(* IEC 61131-3 sources: moqui-plc/simatic-ax/src/moqui/framework/src/main/org/moqui/device, 20 files *)

(* ---- ActuatorActuationType.st ---- *)
TYPE ActuatorActuationType : (
    SingleActuation, (* Single Actuation: Uses enable output only *)
    DoubleActuation, (* Double Actuation: enable/disable are pulses *)
    DoubleActuationNoRetain (* Double Actuation: enable/disable are levels *)
); END_TYPE

(* ---- ActuatorFeedbackType.st ---- *)
TYPE ActuatorFeedbackType : (
	WithoutFeedback, (* No feedback *)
    SingleDisableFeedback, (* Single Deactivation Feedback: Only disabledSensor *)
    SingleEnableFeedback, (* Single Activation Feedback: Only enabledSensor *)
	DoubleFeedback (* Double Feedback: Both sensors *)
); END_TYPE

(* ---- ActuatorModel.st ---- *)
TYPE ActuatorModel : (
	ABBACH580, (* ABB ACH580 *)
	CTM700, (* Control Techniques CM700 *)
	DanfossFC102, (* Danfoss FC102 *)
	ABBPSTX (* ABB PSTX SoftStarter *)
	(* etc. *)
); END_TYPE

(* ---- ActuatorStatus.st ---- *)
TYPE ActuatorStatus : (
	Disabled, (* Stable *)
	EnablePhase, (* Unstable *)
	Enabled, (* Stable *)
	DisablePhase (* Unstable *)
); END_TYPE

(* ---- ActuatorType.st ---- *)
TYPE ActuatorType : (
  OnOff, (* Fallback value *)
  Contactor,
  SoftStarter,
  Vfd, (* Frequency converter / Inverter drive *)
  PneumaticCylinder,
  PneumaticValve,
  HydraulicCylinder,
  HydraulicValve,
  Damper,
  SolenoidValve
  (* etc. *)
); END_TYPE

(* ---- DeviceConfigCmdType.st ---- *)
(* After each creation, saving or deletion of device config it will be necessary to reload the config list with the Init command. *)
TYPE DeviceConfigCmdType : (
    Init, (* Init the recipe management component *)
	Create,
    Save,
	Load,
	Delete,
	Reset
); END_TYPE

(* ---- DeviceConfigMgmtStatus.st ---- *)
TYPE DeviceConfigMgmtStatus : (
    Idle,
	Init,
	Resetting,
    Check,
    Load,
    WaitLoad,
    WaitProcessing,
    IncrementIndex,
    Completed,
    Error
); END_TYPE

(* ---- DriveControlWord.st ---- *)
(* Drive control words *)
(* Relevant control word for start, stop and reset commands *)
TYPE DriveControlWord : (
	(* ABB ACS580, ACH580 drive *)
	ABBACH580Reset,
	ABBACH580Stop,
	ABBACH580Start,
	(* Control Techniques M600 drive *)
	CTM600Reset,
	CTM600Stop,
	CTM600Start,
	(* Danfoss FC102 drive *)
	DanfossFC102Reset,
	DanfossFC102Stop,
	DanfossFC102Start
); END_TYPE

(* ---- EdgeTriggerStatus.st ---- *)
TYPE EdgeTriggerStatus : (
	Dormant,
	Executing,
	Done,
	Aborting,
	Aborted,
	Resetting,
	Error
); END_TYPE

(* ---- LevelCtrlStatus.st ---- *)
TYPE LevelCtrlStatus : (
	Dormant,
	Executing,
	Done,
	Aborting,
	Resetting,
	Error
); END_TYPE

(* ---- OperatingMode.st ---- *)
TYPE OperatingMode : (
	Init,
	Run
); END_TYPE

(* ---- RampType.st ---- *)
TYPE RampType : (
    Linear, // Linear ramp.
    SShaped, // S-Shaped ramp.
    Exponential, // Exponential ramp
    Custom // Custom-defined ramp function
); END_TYPE

(* ---- SpeedSetpointLevel.st ---- *)
(* Constants are defined to represent the different speed levels required by a motor.
 * Alternatively, the speed setpoint/reference can be defined as a continuous analog output.
 * It is possible to apply the same logic to other variables such as:
 *     acceleration/deceleration, torque, etc.
 *)
TYPE SpeedSetpointLevel : (
	ZeroSpeed,
	NominalSpeed,
	MinSpeed,
	MaxSpeed,
	JoggingSpeed,
	SafelyLimitedSpeed
	(* etc. *)
); END_TYPE

(* ---- ParseRecipeTime.st ---- *)
USING System.Strings;

FUNCTION ParseRecipeTime : TIME
	VAR_INPUT
		value : STRING;
	END_VAR
	VAR_TEMP
		normalizedValue : STRING[32];
		numberText : STRING[16];
		unitText : STRING[2];
		valueLength : INT;
		magnitude : DINT;
		position : DINT;
	END_VAR

	normalizedValue := value;
	valueLength := LengthOf(normalizedValue);

	IF (valueLength >= INT#5) AND (Substring(normalizedValue, INT#1, INT#5) = 'TIME#') THEN
		normalizedValue := Substring(normalizedValue, INT#6, valueLength - INT#5);
	ELSIF (valueLength >= INT#2) AND (Substring(normalizedValue, INT#1, INT#2) = 'T#') THEN
		normalizedValue := Substring(normalizedValue, INT#3, valueLength - INT#2);
	END_IF;

	valueLength := LengthOf(normalizedValue);
	IF valueLength <= INT#0 THEN
		RETURN;
	END_IF;

	IF (valueLength >= INT#2) AND (Substring(normalizedValue, valueLength - INT#1, INT#2) = 'ms') THEN
		unitText := 'ms';
		numberText := Substring(normalizedValue, INT#1, valueLength - INT#2);
	ELSIF (valueLength >= INT#1) THEN
		unitText := Substring(normalizedValue, valueLength, INT#1);
		numberText := Substring(normalizedValue, INT#1, valueLength - INT#1);
	END_IF;

	magnitude := ParseRecipeDInt(numberText);
	IF magnitude <= DINT#0 THEN
		RETURN;
	END_IF;

	CASE unitText OF
		'ms' :
			FOR position := DINT#1 TO magnitude DO
				ParseRecipeTime := ParseRecipeTime + T#1ms;
			END_FOR;
		's' :
			FOR position := DINT#1 TO magnitude DO
				ParseRecipeTime := ParseRecipeTime + T#1s;
			END_FOR;
		'm' :
			FOR position := DINT#1 TO magnitude DO
				ParseRecipeTime := ParseRecipeTime + T#1m;
			END_FOR;
		'h' :
			FOR position := DINT#1 TO magnitude DO
				ParseRecipeTime := ParseRecipeTime + T#1h;
			END_FOR;
	END_CASE;
END_FUNCTION

(* ---- Actuator.st ---- *)
(*
 * Generic binary actuator control system/automata, including mechanisms diagnostics.
 * In nominal conditions, a binary actuator has only two stable equilibrium states: Disabled, Enabled.
 * It also has two unstable transient states: EnablePhase, DisablePhase.
 * The remainder are inadmissible states that must be detected based on timing conditions.
 * Nominal trajectory in the state space, i.e. the evolution of the state in nominal working conditions:
 *     Disabled --> EnablePhase --> Enabled --> DisabledPhase --> back to Disabled
 * Admissible states transitions:
 *     EnablePhase --> DisablePhase, DisablePhase --> EnablePhase
 *
 * Handshake-based actuator control via VAR_IN_OUT.
 * This function block utilizes a Request/Acknowledge (Handshake) mechanism
 * through VAR_IN_OUT variables to manage asynchronous device operations.
 *
 * Usage Logic:
 *  - The caller sets the 'enableRequest' variable to TRUE to initiate the process.
 *  - The FB monitors this variable and attempts to enable the physical device.
 *  - Upon successful activation, the FB internally resets 'enableRequest' to FALSE.
 *
 * Sequencing and diagnostics:
 *  - Sequencing: By monitoring the falling edge of the request variable (Request -> FALSE),
 *    the application logic can deterministically trigger the next step in a sequence
 *    without relying on timers or intermediate state flags.
 *  - Real-Time diagnostics: If the request remains TRUE beyond a defined timeout period,
 *    it indicates a failure in the handshake (e.g., hardware interlock or communication error).
 *    This allows for immediate error detection (machineError) and prevents the
 *    sequence from advancing in an unsafe state.
 *
 * Note:
 * Since the variable is passed by reference (VAR_IN_OUT), both the caller and
 * the FB share the same memory location, ensuring atomic-like synchronization of the command status.
 * This mechanism is used to allow sequencing of the start/stop phases in the presence of a group of devices.
 *
 *)
FUNCTION_BLOCK Actuator
	(* Request/Ack commands *)
	VAR_IN_OUT
	    enableRequest : BOOL;
	    disableRequest : BOOL;
	END_VAR
	VAR_INPUT
		(* Actuator metadata for logging purpose *)
		actuatorId : STRING;
		actuatorName : STRING;
	  	actuationType : ActuatorActuationType;
		feedbackType : ActuatorFeedbackType;
		model : ActuatorModel;
	    operationType : OperatingMode := OperatingMode#Run;
		(* Clock for diagnosis and fault detection under static and dynamic conditions *)
	    clock : BOOL;
		(* Time limit for the enable/disable phase *)
	    enableTime : UINT;
	    disableTime : UINT;
		(* Preset/Reset *)
	    enablePreset : BOOL := FALSE;
	    (* Enable diagnostics *)
	    diagnosticsEnable : BOOL := TRUE;
	END_VAR
	VAR_INPUT
		(* Actuator status sensors *)
	    enabledSensor : BOOL;
	    disabledSensor : BOOL;
		(* External fault signal (e.g. motor branch-circuit protection, thermal relay) *)
		externalFault : BOOL;
		(* Optional parameters  *)
	  	referenceValue : REAL;
	  	feedback : REAL;
	END_VAR
	VAR_OUTPUT
		(* Diagnostics and fault signals *)
	    fault : BOOL;
	    actuatorFault : BOOL;
	    enabledSensorFault : BOOL;
	    disabledSensorFault : BOOL;
	    notInitialized : BOOL;
		(* Logger name for centralized signal management *)
		loggerName : STRING;
	END_VAR
	VAR_OUTPUT
		(* Output signals *)
		enable : BOOL;
	    disable : BOOL;
	END_VAR
	VAR
	    status : ActuatorStatus;
	    timer : UINT;
	    timeout : BOOL;
		(* Internal logical feedback signals (derived from external sensors and/or state + timeout). *)
		enabled : BOOL;
		disabled : BOOL;
		(* Logger facade *)
		logger : LoggerFacade;
	END_VAR

	(* Initialization handler *)
	IF operationType = OperatingMode#Init THEN
		(* Args validation *)
		IF (actuatorId = '' AND actuatorName = '') THEN
			notInitialized := TRUE;
			RETURN;
		END_IF;

		(* Logger facade init *)
		loggerName := actuatorName;
		IF loggerName = '' THEN
			loggerName := actuatorId;
		END_IF;
		logger.enable := TRUE; logger.loggerName := loggerName;

		logger(message := 'Actuator initialization.', level := LogLevel#DEBUG);

		(* Pre-elaborations for initialization (polymorphism on feedback typology). *)
		CASE feedbackType OF
			ActuatorFeedbackType#DoubleFeedback :
				enabled := enabledSensor;
				disabled := disabledSensor;

			ActuatorFeedbackType#SingleEnableFeedback :
				enabled := enabledSensor;
				disabled := NOT enabled;

			ActuatorFeedbackType#SingleDisableFeedback :
				disabled := disabledSensor;
				enabled := NOT disabled;

			ActuatorFeedbackType#WithoutFeedback :
				enabled := enablePreset;
				disabled := NOT enabled;
		END_CASE;

		enableRequest := FALSE;
		disableRequest := FALSE;

	    IF enablePreset THEN
			logger(message := 'Actuator preset to enabled status.', level := LogLevel#DEBUG);
			enable := TRUE;
			timer := enableTime;

			IF enabled THEN
				status := ActuatorStatus#Enabled;
				notInitialized := FALSE;
			ELSE
				status := ActuatorStatus#EnablePhase;
	            notInitialized := TRUE;
			END_IF;
	    ELSE
			logger(message := 'Actuator preset to disabled status.', level := LogLevel#DEBUG);
			enable := FALSE;
			timer := disableTime;

			IF disabled THEN
	            status := ActuatorStatus#Disabled;
	            notInitialized := FALSE;
	        ELSE
	            status := ActuatorStatus#DisablePhase;
	            notInitialized := TRUE;
	        END_IF;
		END_IF;
	END_IF;

	IF notInitialized THEN logger(message := 'Actuator not initialized.', level := LogLevel#ERROR); END_IF;

	logger(message := 'Running actuator.', level := LogLevel#DEBUG);

	(* Clock handler for diagnosis oriented timing *)
	IF clock AND (timer > UINT#0) THEN
	    timer := timer - UINT#1;
	END_IF;

	(* Timeout computation *)
	timeout := (timer = UINT#0);

	(* Pre-elaborations for feedback polymorphism. *)
	CASE feedbackType OF
		ActuatorFeedbackType#DoubleFeedback :
			enabled := enabledSensor;
			disabled := disabledSensor;

		ActuatorFeedbackType#SingleDisableFeedback :
			disabled := disabledSensor;
			enabled := (NOT disabled) AND ((status = ActuatorStatus#Enabled)
				OR ((status = ActuatorStatus#EnablePhase) AND timeout));

		ActuatorFeedbackType#SingleEnableFeedback :
			enabled := enabledSensor;
			disabled := (NOT enabled) AND ((status = ActuatorStatus#Disabled)
				OR ((status = ActuatorStatus#DisablePhase) AND timeout));

		ActuatorFeedbackType#WithoutFeedback :
			enabled := (status = ActuatorStatus#Enabled) OR ((status = ActuatorStatus#EnablePhase) AND timeout);
			disabled := (status = ActuatorStatus#Disabled) OR ((status = ActuatorStatus#DisablePhase) AND timeout);
	END_CASE;

	(* Generic actuator FSM implementation. *)
	CASE status OF
		ActuatorStatus#Disabled :
			logger(message := 'Actuator disabled.', level := LogLevel#DEBUG);
			disableRequest := FALSE;

			IF enableRequest THEN
				logger(message := 'The actuator received an enable request.', level := LogLevel#DEBUG);
				enable := TRUE;
				timer := enableTime;
				status := ActuatorStatus#EnablePhase;
			END_IF;

		ActuatorStatus#EnablePhase :
			logger(message := 'Actuator in the enabling phase.', level := LogLevel#DEBUG);

			(* Admissible transition: EnablePhase --> DisablePhase *)
			IF disableRequest THEN
				logger(message := 'The actuator received a disable request.', level := LogLevel#DEBUG);
				enableRequest := FALSE;
				enable := FALSE;
				timer := disableTime;
				status := ActuatorStatus#DisablePhase;
			ELSIF enabled THEN
				(* End of the enable phase, by feedback or by timeout in no-feedback typology. *)
				enableRequest := FALSE;
				timer := UINT#0;
				status := ActuatorStatus#Enabled;
			END_IF;

		ActuatorStatus#Enabled :
			logger(message := 'Actuator enabled.', level := LogLevel#DEBUG);
			enableRequest := FALSE;

			IF disableRequest THEN
				logger(message := 'The actuator received a disable request.', level := LogLevel#DEBUG);
				enable := FALSE;
				timer := disableTime;
				status := ActuatorStatus#DisablePhase;
			END_IF;

		ActuatorStatus#DisablePhase :
			logger(message := 'Actuator in the disabling phase.', level := LogLevel#DEBUG);

			(* Admissible transition: DisablePhase --> EnablePhase *)
			IF enableRequest THEN
					logger(message := 'The actuator received an enable request.', level := LogLevel#DEBUG);
					disableRequest := FALSE;
					enable := TRUE;
					timer := enableTime;
					status := ActuatorStatus#EnablePhase;
			ELSIF disabled THEN
				(* End of the disable phase, by feedback or by timeout in no-feedback typology. *)
				disableRequest := FALSE;
				timer := UINT#0;
				status := ActuatorStatus#Disabled;
			END_IF;
	END_CASE;

	(*
	 * Diagnostics handler.
	 * Generation of diagnosis information and fault signals: Detectable faults in dynamic and static conditions.
	 *)
	disabledSensorFault := diagnosticsEnable AND (
	    (NOT enable AND NOT disabled AND NOT enabled
		OR enable AND disabled AND enabled) AND timeout);
	enabledSensorFault := diagnosticsEnable AND (
	    (NOT enable AND disabled AND enabled
		OR enable AND NOT disabled AND NOT enabled) AND timeout);
	actuatorFault := diagnosticsEnable AND (
	    (NOT enable AND NOT disabled AND enabled
		OR enable AND disabled AND NOT enabled) AND timeout);
	fault := disabledSensorFault OR enabledSensorFault OR actuatorFault OR externalFault;
	(* Log faults *)
	IF fault THEN logger(message := 'Fault diagnostics:', level := LogLevel#ERROR); END_IF;
	IF disabledSensorFault THEN logger(message := 'Disabled sensor fault.', level := LogLevel#ERROR); END_IF;
	IF enabledSensorFault THEN logger(message := 'Enabled sensor fault.', level := LogLevel#ERROR); END_IF;
	IF actuatorFault THEN logger(message := 'Actuator fault.', level := LogLevel#ERROR); END_IF;
	IF externalFault THEN logger(message := 'External fault (e.g: Motor branch-circuit protection).', level := LogLevel#ERROR); END_IF;

	(* Post-elaborations for actuation polymorphism. *)
	CASE actuationType OF
		ActuatorActuationType#SingleActuation :
			(* Nothing to do, just use enable *);
		ActuatorActuationType#DoubleActuation :
			disable := NOT enable;
		ActuatorActuationType#DoubleActuationNoRetain :
			enable := enable AND (status = ActuatorStatus#EnablePhase);
			disable := NOT enable AND (status = ActuatorStatus#DisablePhase);
	END_CASE;
	END_FUNCTION_BLOCK

(* ---- DeviceConfigCmds.st ---- *)
USING Siemens.Simatic.S71500.FileAccess;
USING System.Strings;

FUNCTION_BLOCK DeviceConfigCmds
	VAR_EXTERNAL CONSTANT
		DEVICE_CONFIG_LIST_MAX_SIZE : UINT;
		defaultConfigType : STRING;
		deviceConfigStoragePath : STRING;
	END_VAR
	VAR_EXTERNAL
		dev : DeviceFacade;
	END_VAR
	VAR_INPUT
	    configType : STRING := defaultConfigType; (* If empty, set default device config type *)
		(*
	     * The default file name of a recipe is: <configName>.<configType>.<extension>
	     * Device config ID or name used by the commands.
	     *)
	    configName : STRING := '';
	    cmd : DeviceConfigCmdType := DeviceConfigCmdType#Load;
	END_VAR
	VAR_OUTPUT
		(* Device config list *)
		configNameList : ARRAY[0..DEVICE_CONFIG_LIST_MAX_SIZE] OF STRING;
		configNameListSize : UINT;
		error : BOOL;
		errorId : DWORD; (* 16#5000 : InvalidArgs *)
	END_VAR
	VAR
		indexReader : ReadFile;
		recipeReader : ReadFile;
		indexBuffer : ARRAY[0..4095] OF BYTE;
		recipeBuffer : ARRAY[0..16383] OF BYTE;
		configFileNameList : ARRAY[0..DEVICE_CONFIG_LIST_MAX_SIZE] OF STRING;
		activeRecipeFileName : STRING;
		lastConfigName : STRING;
		lastCmd : DeviceConfigCmdType := DeviceConfigCmdType#Reset;
		indexReaderIssued : BOOL;
		recipeReaderIssued : BOOL;
		indexLoaded : BOOL;
		recipeLoaded : BOOL;
		(* Logger facade *)
		logger : LoggerFacade;
	END_VAR
	VAR_TEMP
		listIndex : UINT;
		parseIndex : DINT;
		lineStart : DINT;
		lineEnd : DINT;
		lineLength : DINT;
		tempLength : INT;
		firstSeparator : INT;
		secondSeparator : INT;
		secondSeparatorRelative : INT;
		paramId : DINT;
		componentIndex : DINT;
		commandChanged : BOOL;
		lineText : STRING[254];
		fieldA : STRING[120];
		fieldB : STRING[120];
		fieldC : STRING[120];
		sortTempName : STRING;
		sortTempFileName : STRING;
		sortSwapped : BOOL;
	END_VAR

	VAR CONSTANT
		ERR_INVALID_ARGS : DWORD := DWORD#16#5000;
		ERR_READ_INDEX : DWORD := DWORD#16#5001;
		ERR_PARSE_INDEX : DWORD := DWORD#16#5002;
		ERR_CONFIG_NOT_FOUND : DWORD := DWORD#16#5003;
		ERR_READ_RECIPE : DWORD := DWORD#16#5004;
		ERR_PARSE_RECIPE : DWORD := DWORD#16#5005;
		ERR_NOT_SUPPORTED : DWORD := DWORD#16#5006;
		INDEX_FILE_PATH : STRING := 'UserFiles/index.csv';
		USER_FILES_PREFIX : STRING := 'UserFiles/';
	END_VAR

	(* Logger facade init *)
	logger.enable := TRUE;
	logger.loggerName := 'DeviceConfigCmds';

	commandChanged := (cmd <> lastCmd) OR ((cmd = DeviceConfigCmdType#Load) AND (configName <> lastConfigName));
	IF commandChanged THEN
		indexReaderIssued := FALSE;
		recipeReaderIssued := FALSE;
		indexLoaded := FALSE;
		recipeLoaded := FALSE;
		activeRecipeFileName := '';
		lastCmd := cmd;
		lastConfigName := configName;
	END_IF;

	(* Args validation *)
	IF (configType = '') OR ((cmd <> DeviceConfigCmdType#Init) AND (cmd <> DeviceConfigCmdType#Reset) AND (configName = '')) THEN
		logger(message := 'Invalid arguments.', level := LogLevel#Error);
		error := TRUE;
		errorId := ERR_INVALID_ARGS;
		RETURN;
	END_IF;

	CASE cmd OF
		DeviceConfigCmdType#Init :
			IF commandChanged THEN
				logger(message := 'Loading device config list.');
				listIndex := UINT#0;
				WHILE listIndex <= DEVICE_CONFIG_LIST_MAX_SIZE DO
					configNameList[listIndex] := '';
					configFileNameList[listIndex] := '';
					listIndex := listIndex + UINT#1;
				END_WHILE;
				configNameListSize := UINT#0;
			END_IF;

			indexReader(
				execute := NOT indexReaderIssued AND NOT indexLoaded,
				path := INDEX_FILE_PATH,
				offset := UDINT#0,
				length := UDINT#4096,
				data := indexBuffer
			);
			IF NOT indexReaderIssued AND NOT indexLoaded THEN
				indexReaderIssued := TRUE;
			END_IF;

			IF indexReader.error THEN
				logger(message := 'Error loading device config list from file system.', level := LogLevel#Error);
				error := TRUE;
				errorId := ERR_READ_INDEX;
				RETURN;
			END_IF;

			IF indexReader.busy AND NOT indexReader.done THEN
				error := FALSE;
				errorId := TO_DWORD(indexReader.status);
				RETURN;
			END_IF;

			IF indexReader.done AND NOT indexLoaded THEN
				indexLoaded := TRUE;
				lineStart := DINT#0;

				WHILE lineStart < TO_DINT(indexReader.resultLength) DO
					WHILE (lineStart < TO_DINT(indexReader.resultLength))
							AND ((indexBuffer[lineStart] = BYTE#10) OR (indexBuffer[lineStart] = BYTE#13)) DO
						lineStart := lineStart + DINT#1;
					END_WHILE;

					IF lineStart >= TO_DINT(indexReader.resultLength) THEN
						EXIT;
					END_IF;

					lineEnd := lineStart;
					WHILE (lineEnd < TO_DINT(indexReader.resultLength))
							AND (indexBuffer[lineEnd] <> BYTE#10)
							AND (indexBuffer[lineEnd] <> BYTE#13) DO
						lineEnd := lineEnd + DINT#1;
					END_WHILE;

					lineLength := lineEnd - lineStart;
					IF lineLength > DINT#0 THEN
						CharsToString(chars := indexBuffer, startPosition := lineStart, length := TO_UINT(lineLength), result => lineText);
						IF lineText <> 'name,configType,fileName' THEN
							firstSeparator := PositionOf(lineText, ',');
							IF firstSeparator = INT#0 THEN
								error := TRUE;
								errorId := ERR_PARSE_INDEX;
								logger(message := 'Invalid index.csv line.', level := LogLevel#Error);
								RETURN;
							END_IF;

							fieldA := Substring(lineText, INT#1, firstSeparator - INT#1);
							tempLength := LengthOf(lineText);
							fieldB := Substring(lineText, firstSeparator + INT#1, tempLength - firstSeparator);
							secondSeparatorRelative := PositionOf(fieldB, ',');
							IF secondSeparatorRelative = INT#0 THEN
								error := TRUE;
								errorId := ERR_PARSE_INDEX;
								logger(message := 'Invalid index.csv line.', level := LogLevel#Error);
								RETURN;
							END_IF;

							fieldC := Substring(fieldB, secondSeparatorRelative + INT#1, LengthOf(fieldB) - secondSeparatorRelative);
							fieldB := Substring(fieldB, INT#1, secondSeparatorRelative - INT#1);

							IF fieldB = configType THEN
								IF configNameListSize <= DEVICE_CONFIG_LIST_MAX_SIZE THEN
									configNameList[configNameListSize] := fieldA;
									configFileNameList[configNameListSize] := fieldC;
									configNameListSize := configNameListSize + UINT#1;
								END_IF;
							END_IF;
						END_IF;
					END_IF;

					lineStart := lineEnd + DINT#1;
				END_WHILE;

				IF configNameListSize > UINT#1 THEN
					REPEAT
						sortSwapped := FALSE;
						parseIndex := DINT#0;
						WHILE parseIndex < TO_DINT(configNameListSize - UINT#1) DO
							IF configNameList[TO_UINT(parseIndex)] > configNameList[TO_UINT(parseIndex + DINT#1)] THEN
								sortTempName := configNameList[TO_UINT(parseIndex)];
								configNameList[TO_UINT(parseIndex)] := configNameList[TO_UINT(parseIndex + DINT#1)];
								configNameList[TO_UINT(parseIndex + DINT#1)] := sortTempName;

								sortTempFileName := configFileNameList[TO_UINT(parseIndex)];
								configFileNameList[TO_UINT(parseIndex)] := configFileNameList[TO_UINT(parseIndex + DINT#1)];
								configFileNameList[TO_UINT(parseIndex + DINT#1)] := sortTempFileName;
								sortSwapped := TRUE;
							END_IF;
							parseIndex := parseIndex + DINT#1;
						END_WHILE;
					UNTIL NOT sortSwapped
					END_REPEAT;
				END_IF;
			END_IF;

			error := FALSE;
			errorId := DWORD#16#0000;

		DeviceConfigCmdType#Load :
			activeRecipeFileName := '';
			parseIndex := DINT#0;
			WHILE parseIndex < TO_DINT(configNameListSize) DO
				IF configNameList[TO_UINT(parseIndex)] = configName THEN
					activeRecipeFileName := configFileNameList[TO_UINT(parseIndex)];
				END_IF;
				parseIndex := parseIndex + DINT#1;
			END_WHILE;

			IF activeRecipeFileName = '' THEN
				error := TRUE;
				errorId := ERR_CONFIG_NOT_FOUND;
				logger(message := 'Device config not found in index.', level := LogLevel#Error);
				RETURN;
			END_IF;

			recipeReader(
				execute := NOT recipeReaderIssued AND NOT recipeLoaded,
				path := Concat(USER_FILES_PREFIX, activeRecipeFileName),
				offset := UDINT#0,
				length := UDINT#16384,
				data := recipeBuffer
			);
			IF NOT recipeReaderIssued AND NOT recipeLoaded THEN
				recipeReaderIssued := TRUE;
			END_IF;

			IF recipeReader.error THEN
				logger(message := 'Error loading device config recipe file.', level := LogLevel#Error);
				error := TRUE;
				errorId := ERR_READ_RECIPE;
				RETURN;
			END_IF;

			IF recipeReader.busy AND NOT recipeReader.done THEN
				error := FALSE;
				errorId := TO_DWORD(recipeReader.status);
				RETURN;
			END_IF;

			IF recipeReader.done AND NOT recipeLoaded THEN
				recipeLoaded := TRUE;
				lineStart := DINT#0;

				WHILE lineStart < TO_DINT(recipeReader.resultLength) DO
					WHILE (lineStart < TO_DINT(recipeReader.resultLength))
							AND ((recipeBuffer[lineStart] = BYTE#10) OR (recipeBuffer[lineStart] = BYTE#13)) DO
						lineStart := lineStart + DINT#1;
					END_WHILE;

					IF lineStart >= TO_DINT(recipeReader.resultLength) THEN
						EXIT;
					END_IF;

					lineEnd := lineStart;
					WHILE (lineEnd < TO_DINT(recipeReader.resultLength))
							AND (recipeBuffer[lineEnd] <> BYTE#10)
							AND (recipeBuffer[lineEnd] <> BYTE#13) DO
						lineEnd := lineEnd + DINT#1;
					END_WHILE;

					lineLength := lineEnd - lineStart;
					IF lineLength > DINT#0 THEN
						CharsToString(chars := recipeBuffer, startPosition := lineStart, length := TO_UINT(lineLength), result => lineText);
						firstSeparator := PositionOf(lineText, ';');
						IF firstSeparator = INT#0 THEN
							error := TRUE;
							errorId := ERR_PARSE_RECIPE;
							logger(message := 'Invalid AX recipe line.', level := LogLevel#Error);
							RETURN;
						END_IF;

						fieldA := Substring(lineText, INT#1, firstSeparator - INT#1);
						tempLength := LengthOf(lineText);
						fieldB := Substring(lineText, firstSeparator + INT#1, tempLength - firstSeparator);
						secondSeparatorRelative := PositionOf(fieldB, ';');
						IF secondSeparatorRelative = INT#0 THEN
							error := TRUE;
							errorId := ERR_PARSE_RECIPE;
							logger(message := 'Invalid AX recipe line.', level := LogLevel#Error);
							RETURN;
						END_IF;

						fieldC := Substring(fieldB, secondSeparatorRelative + INT#1, LengthOf(fieldB) - secondSeparatorRelative);
						fieldB := Substring(fieldB, INT#1, secondSeparatorRelative - INT#1);
						paramId := ParseRecipeDInt(fieldA);

						CASE paramId OF
							DINT#1 : dev.tempSetpoint := ParseRecipeReal(fieldC);
							DINT#2 : dev.tempHysteresis := ParseRecipeReal(fieldC);
							DINT#3 : dev.tempMin := ParseRecipeReal(fieldC);
							DINT#4 : dev.tempMax := ParseRecipeReal(fieldC);
							DINT#5 : dev.rhSetpoint := ParseRecipeReal(fieldC);
							DINT#6 : dev.rhHysteresis := ParseRecipeReal(fieldC);
							DINT#7 : dev.rhMin := ParseRecipeReal(fieldC);
							DINT#8 : dev.rhMax := ParseRecipeReal(fieldC);
							DINT#9 : dev.airDistributionEnabled := (fieldC = 'TRUE');
							DINT#10 : dev.setPointTimeHigh := TO_UINT(ParseRecipeDInt(fieldC));
							DINT#11 : dev.setPointTimeLow := TO_UINT(ParseRecipeDInt(fieldC));
							DINT#14 : dev.ductTempMin := ParseRecipeReal(fieldC);
							DINT#15 : dev.ductTempMax := ParseRecipeReal(fieldC);
							DINT#16 : dev.ductRhMax := ParseRecipeReal(fieldC);
							DINT#17 : dev.rhControlEnabled := (fieldC = 'TRUE');
							DINT#18 : dev.rhControlOnly := (fieldC = 'TRUE');
							DINT#20 : dev.airMixingEnabled := (fieldC = 'TRUE');
							DINT#21 : dev.estimatedRuntime := TO_UDINT(ParseRecipeDInt(fieldC));
							DINT#22 : dev.minRuntime := TO_UDINT(ParseRecipeDInt(fieldC));
							DINT#23 : dev.estimatedBreakDuration := TO_UDINT(ParseRecipeDInt(fieldC));
							DINT#24 : dev.minBreakDuration := TO_UDINT(ParseRecipeDInt(fieldC));
							DINT#25 : dev.processEstimatedDuration := TO_UDINT(ParseRecipeDInt(fieldC));
							DINT#26 : dev.processMinDuration := TO_UDINT(ParseRecipeDInt(fieldC));
							DINT#27 : dev.airFlowRef := ParseRecipeReal(fieldC);
							DINT#28 : dev.ahuFanSpeedSetpoint := ParseRecipeReal(fieldC);
							DINT#29 : dev.tempFeedback := ParseRecipeReal(fieldC);
							DINT#30 : dev.rhFeedback := ParseRecipeReal(fieldC);
							DINT#33 : dev.ductTempFeedback := ParseRecipeReal(fieldC);
							DINT#34 : dev.ductRhFeedback := ParseRecipeReal(fieldC);
							DINT#35 : dev.coldGlycolPump.actuatorId := fieldC;
							DINT#36 : dev.coldGlycolPump.actuatorName := fieldC;
							DINT#37 :
								CASE ParseRecipeDInt(fieldC) OF
									DINT#0 : dev.coldGlycolPump.actuationType := ActuatorActuationType#SingleActuation;
									DINT#1 : dev.coldGlycolPump.actuationType := ActuatorActuationType#DoubleActuation;
									DINT#2 : dev.coldGlycolPump.actuationType := ActuatorActuationType#DoubleActuationNoRetain;
								END_CASE;
							DINT#38 :
								CASE ParseRecipeDInt(fieldC) OF
									DINT#0 : dev.coldGlycolPump.feedbackType := ActuatorFeedbackType#WithoutFeedback;
									DINT#1 : dev.coldGlycolPump.feedbackType := ActuatorFeedbackType#SingleDisableFeedback;
									DINT#2 : dev.coldGlycolPump.feedbackType := ActuatorFeedbackType#SingleEnableFeedback;
									DINT#3 : dev.coldGlycolPump.feedbackType := ActuatorFeedbackType#DoubleFeedback;
								END_CASE;
							DINT#39 :
								CASE ParseRecipeDInt(fieldC) OF
									DINT#0 : dev.coldGlycolPump.model := ActuatorModel#ABBACH580;
									DINT#1 : dev.coldGlycolPump.model := ActuatorModel#CTM700;
									DINT#2 : dev.coldGlycolPump.model := ActuatorModel#DanfossFC102;
									DINT#3 : dev.coldGlycolPump.model := ActuatorModel#ABBPSTX;
								END_CASE;
							DINT#40 : dev.coldGlycolPump.enableTime := TO_UINT(ParseRecipeDInt(fieldC));
							DINT#41 : dev.coldGlycolPump.disableTime := TO_UINT(ParseRecipeDInt(fieldC));
							DINT#42 : dev.coldGlycolPump.diagnosticsEnable := (fieldC = 'TRUE');
							DINT#43 : dev.hotGlycolPump.actuatorId := fieldC;
							DINT#44 : dev.hotGlycolPump.actuatorName := fieldC;
							DINT#45 :
								CASE ParseRecipeDInt(fieldC) OF
									DINT#0 : dev.hotGlycolPump.actuationType := ActuatorActuationType#SingleActuation;
									DINT#1 : dev.hotGlycolPump.actuationType := ActuatorActuationType#DoubleActuation;
									DINT#2 : dev.hotGlycolPump.actuationType := ActuatorActuationType#DoubleActuationNoRetain;
								END_CASE;
							DINT#46 :
								CASE ParseRecipeDInt(fieldC) OF
									DINT#0 : dev.hotGlycolPump.feedbackType := ActuatorFeedbackType#WithoutFeedback;
									DINT#1 : dev.hotGlycolPump.feedbackType := ActuatorFeedbackType#SingleDisableFeedback;
									DINT#2 : dev.hotGlycolPump.feedbackType := ActuatorFeedbackType#SingleEnableFeedback;
									DINT#3 : dev.hotGlycolPump.feedbackType := ActuatorFeedbackType#DoubleFeedback;
								END_CASE;
							DINT#47 :
								CASE ParseRecipeDInt(fieldC) OF
									DINT#0 : dev.hotGlycolPump.model := ActuatorModel#ABBACH580;
									DINT#1 : dev.hotGlycolPump.model := ActuatorModel#CTM700;
									DINT#2 : dev.hotGlycolPump.model := ActuatorModel#DanfossFC102;
									DINT#3 : dev.hotGlycolPump.model := ActuatorModel#ABBPSTX;
								END_CASE;
							DINT#48 : dev.hotGlycolPump.enableTime := TO_UINT(ParseRecipeDInt(fieldC));
							DINT#49 : dev.hotGlycolPump.disableTime := TO_UINT(ParseRecipeDInt(fieldC));
							DINT#50 : dev.hotGlycolPump.diagnosticsEnable := (fieldC = 'TRUE');
							DINT#51 : dev.airFlow.actuatorId := fieldC;
							DINT#52 : dev.airFlow.actuatorName := fieldC;
							DINT#53 :
								CASE ParseRecipeDInt(fieldC) OF
									DINT#0 : dev.airFlow.actuationType := ActuatorActuationType#SingleActuation;
									DINT#1 : dev.airFlow.actuationType := ActuatorActuationType#DoubleActuation;
									DINT#2 : dev.airFlow.actuationType := ActuatorActuationType#DoubleActuationNoRetain;
								END_CASE;
							DINT#54 :
								CASE ParseRecipeDInt(fieldC) OF
									DINT#0 : dev.airFlow.feedbackType := ActuatorFeedbackType#WithoutFeedback;
									DINT#1 : dev.airFlow.feedbackType := ActuatorFeedbackType#SingleDisableFeedback;
									DINT#2 : dev.airFlow.feedbackType := ActuatorFeedbackType#SingleEnableFeedback;
									DINT#3 : dev.airFlow.feedbackType := ActuatorFeedbackType#DoubleFeedback;
								END_CASE;
							DINT#55 :
								CASE ParseRecipeDInt(fieldC) OF
									DINT#0 : dev.airFlow.model := ActuatorModel#ABBACH580;
									DINT#1 : dev.airFlow.model := ActuatorModel#CTM700;
									DINT#2 : dev.airFlow.model := ActuatorModel#DanfossFC102;
									DINT#3 : dev.airFlow.model := ActuatorModel#ABBPSTX;
								END_CASE;
							DINT#56 : dev.airFlow.enableTime := TO_UINT(ParseRecipeDInt(fieldC));
							DINT#57 : dev.airFlow.disableTime := TO_UINT(ParseRecipeDInt(fieldC));
							DINT#58 : dev.airFlow.diagnosticsEnable := (fieldC = 'TRUE');
							DINT#59 : dev.coldGlycolValve.controlSystemId := fieldC;
							DINT#60 : dev.coldGlycolValve.controlSystemName := fieldC;
							DINT#61 : dev.coldGlycolValve.gain := ParseRecipeReal(fieldC);
							DINT#62 : dev.coldGlycolValve.integrationTime := ParseRecipeReal(fieldC);
							DINT#63 : dev.coldGlycolValve.derivationTime := ParseRecipeReal(fieldC);
							DINT#64 : dev.coldGlycolValve.setpointMin := ParseRecipeReal(fieldC);
							DINT#65 : dev.coldGlycolValve.setpointMax := ParseRecipeReal(fieldC);
							DINT#66 : dev.coldGlycolValve.outputMin := ParseRecipeReal(fieldC);
							DINT#67 : dev.coldGlycolValve.outputMax := ParseRecipeReal(fieldC);
							DINT#68 : dev.coldGlycolValve.atSetpointHysteresis := ParseRecipeReal(fieldC);
							DINT#69 : dev.coldGlycolValve.tickTime := ParseRecipeTime(fieldC);
							DINT#70 : dev.hotGlycolValve.controlSystemId := fieldC;
							DINT#71 : dev.hotGlycolValve.controlSystemName := fieldC;
							DINT#72 : dev.hotGlycolValve.gain := ParseRecipeReal(fieldC);
							DINT#73 : dev.hotGlycolValve.integrationTime := ParseRecipeReal(fieldC);
							DINT#74 : dev.hotGlycolValve.derivationTime := ParseRecipeReal(fieldC);
							DINT#75 : dev.hotGlycolValve.setpointMin := ParseRecipeReal(fieldC);
							DINT#76 : dev.hotGlycolValve.setpointMax := ParseRecipeReal(fieldC);
							DINT#77 : dev.hotGlycolValve.outputMin := ParseRecipeReal(fieldC);
							DINT#78 : dev.hotGlycolValve.outputMax := ParseRecipeReal(fieldC);
							DINT#79 : dev.hotGlycolValve.atSetpointHysteresis := ParseRecipeReal(fieldC);
							DINT#80 : dev.hotGlycolValve.tickTime := ParseRecipeTime(fieldC);
							DINT#81 : dev.ahuFan.controlSystemId := fieldC;
							DINT#82 : dev.ahuFan.controlSystemName := fieldC;
							DINT#83 : dev.ahuFan.gain := ParseRecipeReal(fieldC);
							DINT#84 : dev.ahuFan.integrationTime := ParseRecipeReal(fieldC);
							DINT#85 : dev.ahuFan.derivationTime := ParseRecipeReal(fieldC);
							DINT#86 : dev.ahuFan.setpointMin := ParseRecipeReal(fieldC);
							DINT#87 : dev.ahuFan.setpointMax := ParseRecipeReal(fieldC);
							DINT#88 : dev.ahuFan.outputMin := ParseRecipeReal(fieldC);
							DINT#89 : dev.ahuFan.outputMax := ParseRecipeReal(fieldC);
							DINT#90 : dev.ahuFan.atSetpointHysteresis := ParseRecipeReal(fieldC);
							DINT#91 : dev.ahuFan.tickTime := ParseRecipeTime(fieldC);
						END_CASE;
					END_IF;

					lineStart := lineEnd + DINT#1;
				END_WHILE;

				logger(message := Concat(Concat(Concat('Loaded device config ', configName), ' of type '), configType));
			END_IF;

			error := FALSE;
			errorId := DWORD#16#0000;

	    DeviceConfigCmdType#Create :
			error := TRUE;
			errorId := ERR_NOT_SUPPORTED;
			logger(message := 'Create is not supported in AX runtime.', level := LogLevel#Error);

	    DeviceConfigCmdType#Save :
	        error := TRUE;
	        errorId := ERR_NOT_SUPPORTED;
			logger(message := 'Save is not supported in AX runtime.', level := LogLevel#Error);

	    DeviceConfigCmdType#Delete :
	        error := TRUE;
			errorId := ERR_NOT_SUPPORTED;
			logger(message := 'Delete is not supported in AX runtime.', level := LogLevel#Error);

		DeviceConfigCmdType#Reset :
			logger(message := 'Resetting device config list.');
			listIndex := UINT#0;
			WHILE listIndex <= DEVICE_CONFIG_LIST_MAX_SIZE DO
				configNameList[listIndex] := '';
				configFileNameList[listIndex] := '';
				listIndex := listIndex + UINT#1;
			END_WHILE;
			configNameListSize := UINT#0;
			indexReaderIssued := FALSE;
			recipeReaderIssued := FALSE;
			indexLoaded := FALSE;
			recipeLoaded := FALSE;
			activeRecipeFileName := '';
			error := FALSE;
			errorId := DWORD#16#0000;
	END_CASE;
END_FUNCTION_BLOCK

(* ---- DeviceConfigMgmt.st ---- *)
(*
 * Pure recipe sequencing logic. Implement complex logic, including micro-recipe composition,
 * alternative recipes, condition-based recipes, etc., if needed.
 *)
FUNCTION_BLOCK DeviceConfigMgmt
	VAR_EXTERNAL CONSTANT
		defaultConfigType : STRING;
	END_VAR
	VAR_INPUT
		enable : BOOL;
		continueAfterError : BOOL;
		configCompleted : BOOL; (* Config processed feedback *)
	END_VAR
	VAR_OUTPUT
	    done, allConfigLoaded, busy, error : BOOL;
		errorId : DWORD;
	END_VAR
	VAR
	    status : DeviceConfigMgmtStatus := DeviceConfigMgmtStatus#Idle;
	    configCmds : DeviceConfigCmds;
	    currentConfigIndex : UINT := UINT#0;
		(* Logger facade *)
	    logger : LoggerFacade;
		init : BOOL;
		configCompletedREdge : R_TRIG;
		configCmdsBusy : BOOL;
	END_VAR

	IF NOT init THEN
		(* Logger facade init *)
		logger.enable := TRUE; logger.loggerName := 'DeviceConfigMgmt';
		init := TRUE;
	END_IF;

	configCompletedREdge(CLK := configCompleted);
	configCmdsBusy := (configCmds.errorId = DWORD#16#7001) OR (configCmds.errorId = DWORD#16#7002);

	CASE status OF
	    DeviceConfigMgmtStatus#Idle :
			done := FALSE; busy := FALSE;

	        IF enable THEN
				busy := TRUE;
				(* Setup the default config type *)
	            configCmds.configType := defaultConfigType;
	            status := DeviceConfigMgmtStatus#Init;
	        END_IF;

	    DeviceConfigMgmtStatus#Init :
			allConfigLoaded := FALSE;
			busy := TRUE;
			configCmds(cmd := DeviceConfigCmdType#Init, error => error, errorId => errorId);

	        IF configCmds.error THEN
				status := DeviceConfigMgmtStatus#Resetting;
			ELSIF configCmdsBusy THEN
				status := DeviceConfigMgmtStatus#Init;
			ELSE
	            status := DeviceConfigMgmtStatus#Load;
	        END_IF;

	    DeviceConfigMgmtStatus#Load :
			busy := TRUE;
	        IF currentConfigIndex >= configCmds.configNameListSize THEN
	            status := DeviceConfigMgmtStatus#Completed;
	        ELSE
	            configCmds.configName := configCmds.configNameList[currentConfigIndex];
	            configCmds(cmd := DeviceConfigCmdType#Load, error => error, errorId => errorId);
	            IF configCmds.error THEN
	                status := DeviceConfigMgmtStatus#Resetting;
	            ELSIF configCmdsBusy THEN
	                status := DeviceConfigMgmtStatus#WaitLoad;
	            ELSE
	                status := DeviceConfigMgmtStatus#WaitProcessing;
	            END_IF;
	        END_IF;

	    DeviceConfigMgmtStatus#WaitLoad :
			done := FALSE;
			busy := TRUE;
	        configCmds.configName := configCmds.configNameList[currentConfigIndex];
	        configCmds(cmd := DeviceConfigCmdType#Load, error => error, errorId => errorId);
	        IF configCmds.error THEN
	            status := DeviceConfigMgmtStatus#Resetting;
	        ELSIF configCmdsBusy THEN
	            status := DeviceConfigMgmtStatus#WaitLoad;
	        ELSE
	            status := DeviceConfigMgmtStatus#WaitProcessing;
	        END_IF;

	    DeviceConfigMgmtStatus#WaitProcessing :
			done := TRUE;
			busy := FALSE;

	        IF configCompletedREdge.Q THEN
	            done := FALSE;
	            logger(message := configCmds.configName);
	            currentConfigIndex := currentConfigIndex + UINT#1;
	            status := DeviceConfigMgmtStatus#Load;
	        END_IF;

	    DeviceConfigMgmtStatus#Completed :
	        allConfigLoaded := TRUE;
			done := TRUE;
			busy := FALSE;
			error := FALSE;
			currentConfigIndex := UINT#0;
	        logger(message := 'All device configs loaded.');
	        status := DeviceConfigMgmtStatus#Idle;

	    DeviceConfigMgmtStatus#Resetting :
	        configCmds(cmd := DeviceConfigCmdType#Reset, error => error, errorId => errorId);
			IF NOT continueAfterError THEN
	        	currentConfigIndex := UINT#0;
	        END_IF;

	        status := DeviceConfigMgmtStatus#Init;
	END_CASE;
	END_FUNCTION_BLOCK

(* ---- EdgeTrigStatusMgr.st ---- *)
(*
Edge triggered status manager.
The PLCOpen standard presents “service/command” function block patterns
that manage the execution of a request (edge-triggered)
or the maintenance of a condition (level-controlled).
The PLCopen patterns model the lifecycle of a command, not the state of the device.
A command handler FB uses the PLCopen (Action) pattern.
The device model maintains the bistable state (Reality/Feedback).
The command requests a device transition, but does not define the device state.
It makes sense to model triggers and levels for physical devices only as an interface contract
between the caller and the device controller, not as the “physical truth” of the device.
An example of edge-triggered functionality is a move-to-position command which,
after being initialized via the input execute, runs till finalized.
For the detection of a rising edge in a function block, two PLC cycles are necessary.
Thus, if the requirement is to be able to process a new value in each cycle, an edge-triggered model cannot serve as a solution.
See the PLCOpen standard document "Creating PLCopen compliant Function Block libraries" for details.

Variant, abort used?, timeLimit, timeout, Behavior
ETrig,       FALSE,       0,        0,    Base: activates on front, ends on readyCondition
ETrigTo,     FALSE,       0,        > 0,  With timeout: if it doesn't finish within timeout, it goes to Error.
ETrigTI,     FALSE,       > 0,      0,    With timeLimit: allows you to divide the work over multiple cycles.
ETrigTITo,   FALSE,       > 0,      > 0,  Complete: both cyclical limit and total timeout management.
ETrigA,      TRUE,        0,        0,    With Aborting: It can be stopped and switched to Aborted.
ETrigATo,    TRUE,        0,        > 0,  With Aborting and timeout: if it doesn't finish within timeout, it goes to Error.
ETrigATI,    TRUE,        > 0,      0,    With Aborting and timeLimit: allows you to divide the work over multiple cycles.
ETrigATITo,  TRUE,        > 0,      > 0,  Complete: both Aborting, cyclical limit and total timeout management.

*)
FUNCTION_BLOCK EdgeTrigStatusMgr
	VAR_INPUT
		(* Initialize and start operation on rising edge and stay active till finalized or aborted. *)
	    execute : BOOL;
	    readyCondition : BOOL; (* Operation completed feedback *)
		(* Interrupt request (ETrigA Variants) to abort the process. *)
	    abortRequest : BOOL;
	    abortComplete : BOOL; (* Aborting feedback *)
	    resetRequest : BOOL; (* Manual reset request *)
	    resetComplete : BOOL; (* Reset feedback *)
	    errorCondition : BOOL; (* Functional error from external logic *)
		(*
		 * PLCOpen: timeLimit (Tl): here the time limit is set that
		 * the operation stays within the cycle time.
		 * In that way a longer operation can be divided over several cycles.
		 *)
	    timeLimit : UINT; (* 0 = inactive *)
		(*
	     * PLCOpen: timeout (To): the overall operating time of the
		 * defined operation should be lower than the time(in μs)
	     * as specified by the input value timeout.
		 * The combination of them both (TlTo) is valid.
	     *)
	    timeout : UINT; (* 0 = inactive *)
	    clock : BOOL; (* Clock signal *)
	END_VAR
	VAR_OUTPUT
	    done : BOOL; (* Operation completed successfully *)
	    busy : BOOL; (* Operation in progress *)
	    error : BOOL; (* Active error *)
	    errorId : INT; (* PLCopen: Error ID. Example 1 = ExternalError, 2 = Timeout *)
	    aborted : BOOL; (* Operation aborted *)
	    activeCycle : BOOL; (* TRUE when the caller needs to execute the logic *)
	END_VAR
	VAR
	    status : EdgeTriggerStatus := EdgeTriggerStatus#Dormant; (* FSM internal status. States: 0- Dormant, 1 - Executing, 2 - Done, 3 - Aborting, 4 - Aborted, 5 - Resetting, 6 - Error *)
	    timeLimitTimer : UINT;
	    timeoutTimer : UINT;
	    prevExecute : BOOL; (* Memory for edge detection *)
	END_VAR

	(* Time management *)
	IF clock THEN
		(* TimeLimit (Tl): cyclic timeslice management *)
		IF timeLimit > UINT#0 AND status = EdgeTriggerStatus#Executing THEN
			IF timeLimitTimer > UINT#0 THEN
				timeLimitTimer := timeLimitTimer - UINT#1;
			ELSE
				(* New invocation timeslice *)
				timeLimitTimer := timeLimit;
			END_IF;
		END_IF;

		(* TimeOut (To): The total timeout only runs during execution *)
		IF timeoutTimer > UINT#0 AND status = EdgeTriggerStatus#Executing THEN
			timeoutTimer := timeoutTimer - UINT#1;
		END_IF;
	END_IF;

	CASE status OF
	    EdgeTriggerStatus#Dormant :
	        done := FALSE; busy := FALSE; aborted := FALSE; error := FALSE; errorId := 0; activeCycle := FALSE;

	        (* Rising edge detection *)
	        IF execute AND NOT prevExecute THEN
	            timeoutTimer := timeout;
				timeLimitTimer := timeLimit;
	            status := EdgeTriggerStatus#Executing;
	        END_IF;

	    EdgeTriggerStatus#Executing :
	        busy := TRUE;
			(* Enable caller logic: active if there is no cycle limit or if the cycle time has not expired. *)
	        activeCycle := (timeLimit = UINT#0) OR (timeLimitTimer > UINT#0);

	        IF errorCondition OR ((timeout > UINT#0) AND (timeoutTimer = UINT#0)) THEN
	            status := EdgeTriggerStatus#Error;
	        ELSIF abortRequest THEN
	            status := EdgeTriggerStatus#Aborting;
	        ELSIF readyCondition THEN
	            status := EdgeTriggerStatus#Done; (* Target achieved *)
	        END_IF;

	    EdgeTriggerStatus#Aborting :
	        activeCycle := FALSE;

	        IF errorCondition OR ((timeout > UINT#0) AND (timeoutTimer = UINT#0)) THEN
	            status := EdgeTriggerStatus#Error;
	        ELSIF abortComplete THEN
				status := EdgeTriggerStatus#Aborted;
			END_IF;

	    EdgeTriggerStatus#Aborted :
	        busy := FALSE; aborted := TRUE;

	        (* Transition to resetting on the falling edge of execute *)
	        IF resetRequest OR NOT execute THEN
				status := EdgeTriggerStatus#Resetting;
			END_IF;

	    EdgeTriggerStatus#Done :
	        busy := FALSE; done := TRUE; activeCycle := FALSE;

			(* Transition to resetting on the falling edge of execute *)
	        IF resetRequest OR NOT execute THEN
				status := EdgeTriggerStatus#Resetting;
			END_IF;

	    EdgeTriggerStatus#Error :
	        busy := FALSE; activeCycle := FALSE; error := TRUE;

	        IF errorCondition THEN
	            errorId := 1; (* ExternalError *)
	        ELSE
	            errorId := 2; (* Total timeout expired *)
	        END_IF;

	        IF resetRequest OR NOT execute THEN
				status := EdgeTriggerStatus#Resetting;
			END_IF;

	    EdgeTriggerStatus#Resetting :
	        done := FALSE; aborted := FALSE; error := FALSE; errorId := 0; activeCycle := FALSE;

			IF resetComplete THEN
				status := EdgeTriggerStatus#Dormant;
			END_IF;
	END_CASE;

	prevExecute := execute;
	END_FUNCTION_BLOCK

(* ---- ProcessPid.st ---- *)
FUNCTION_BLOCK ProcessPid
VAR_INPUT
    enable : BOOL;
    reset : BOOL;
    controlSystemId : STRING;
    controlSystemName : STRING;
    feedback : REAL;
    feedbackMultiplier : REAL := REAL#1.0;
    setpoint : REAL;
    atSetpointHysteresis : REAL;
    setpointMultiplier : REAL := REAL#1.0;
    setpointMin : REAL;
    setpointMax : REAL;
    setpointRampType : RampType := RampType#Linear;
    setpointIncreaseTime : TIME := T#0S;
    setpointDecreaseTime : TIME := T#0S;
    setpointFreezeEnable : BOOL;
    deviationInversion : BOOL;
    outputMin : REAL;
    outputMax : REAL;
    outputFreezeEnable : BOOL;
    gain : REAL := REAL#1.0;
    integrationTime : REAL := REAL#0.0;
    derivationTime : REAL := REAL#0.0;
    offset : REAL := REAL#0.0;
    deadbandRange : REAL;
    deadbandDelay : TIME;
    sleepLevel : REAL := REAL#0.0;
    sleepDelay : TIME;
    wakeupDeviation : REAL;
    wakeupDelay : TIME;
    sleepBoostLevel : REAL := REAL#0.0;
    sleepBoostTime : TIME;
    trackingMode : BOOL := FALSE;
    trackingRef : REAL := REAL#0.0;
    clock : BOOL;
    tickTime : TIME := T#10ms;
    setpointEpsilon : REAL := REAL#0.000001;
END_VAR
VAR_OUTPUT
    feedbackActual : REAL;
    setpointActual : REAL;
    deviationActual : REAL;
    outputActual : REAL;
    invalidConfig : BOOL;
    active : BOOL;
    atSetpoint : BOOL;
    zeroOutput : BOOL;
    setpointFrozen : BOOL;
    outputFrozen : BOOL;
    sleepMode : BOOL;
    sleepBoost : BOOL;
    deadband : BOOL;
    tracking : BOOL;
    outputLimitsActive : BOOL;
    overflow : BOOL;
    loggerName : STRING;
END_VAR
VAR
    deadbandCounter : UDINT;
    sleepCounter : UDINT;
    wakeupCounter : UDINT;
    sleepBoostCounter : UDINT;
    integralTerm : REAL;
    previousDeviation : REAL;
    previousOutput : REAL;
    lastOutput : REAL;
    lastPidOutput : REAL;
    setpointTarget : REAL;
    setpointInternal : REAL;
    lastSetpoint : REAL;
    lastSetpointTarget : REAL;
    prevReset : BOOL;
    resetEdge : BOOL;
    manualMode : BOOL;
    yManual : REAL;
    sleepReq : BOOL;
    wakeupReq : BOOL;
    startRamp : BOOL;
    proportionalTerm : REAL;
    derivativeTerm : REAL;
    deltaDeviation : REAL;
    rawOutput : REAL;
    deviationMagnitude : REAL;
    deltaTime : REAL;
    spRange : REAL;
    increaseTicks : UDINT;
    decreaseTicks : UDINT;
    delayTicks : UDINT;
    rampStep : REAL;
    remainingTime : TIME;
    logger : LoggerFacade;
    sShapedFunc : SShapedFunc;
    expRamp : IIRFilter;
END_VAR

(* controlSystemId is the exact Device.deviceId; controlSystemName is descriptive only. *)
loggerName := controlSystemId;
logger.enable := TRUE;
logger.loggerName := loggerName;

resetEdge := reset AND NOT prevReset;
prevReset := reset;

invalidConfig := FALSE;
overflow := FALSE;
outputLimitsActive := FALSE;
tracking := FALSE;

IF tickTime <= T#0S THEN
    invalidConfig := TRUE;
    active := FALSE;
    outputActual := REAL#0.0;
    RETURN;
END_IF;

IF (gain <= REAL#0.0)
        OR (integrationTime < REAL#0.0)
        OR (derivationTime < REAL#0.0)
        OR (setpointMin > setpointMax)
        OR (outputMin > outputMax) THEN
    invalidConfig := TRUE;
    active := FALSE;
    outputActual := REAL#0.0;
    logger(message := 'Invalid PID configuration.', level := LogLevel#Error);
    RETURN;
END_IF;

IF NOT enable THEN
    active := FALSE;
    atSetpoint := FALSE;
    zeroOutput := TRUE;
    setpointFrozen := FALSE;
    outputFrozen := FALSE;
    sleepMode := FALSE;
    sleepBoost := FALSE;
    deadband := FALSE;
    outputActual := REAL#0.0;
    lastOutput := REAL#0.0;
    previousOutput := REAL#0.0;
    lastPidOutput := REAL#0.0;
    deadbandCounter := UDINT#0;
    sleepCounter := UDINT#0;
    wakeupCounter := UDINT#0;
    sleepBoostCounter := UDINT#0;
    integralTerm := REAL#0.0;
    previousDeviation := REAL#0.0;
    sShapedFunc(execute := FALSE, clock := FALSE);
    expRamp(execute := FALSE, clock := FALSE, reset := TRUE, input := REAL#0.0, T := REAL#0.001);
    RETURN;
END_IF;

active := TRUE;

IF resetEdge THEN
    setpointInternal := REAL#0.0;
    lastSetpoint := REAL#0.0;
    lastSetpointTarget := REAL#0.0;
    previousDeviation := REAL#0.0;
    previousOutput := REAL#0.0;
    lastOutput := REAL#0.0;
    lastPidOutput := REAL#0.0;
    integralTerm := REAL#0.0;
    deadbandCounter := UDINT#0;
    sleepCounter := UDINT#0;
    wakeupCounter := UDINT#0;
    sleepBoostCounter := UDINT#0;
    sleepMode := FALSE;
    sleepBoost := FALSE;
    sShapedFunc(execute := FALSE, clock := FALSE);
    expRamp(execute := FALSE, clock := FALSE, reset := TRUE, input := REAL#0.0, T := REAL#0.001);
    logger(message := 'Reset process PID.', level := LogLevel#Warn);
END_IF;

loggerName := controlSystemId;
logger.loggerName := loggerName;

feedbackActual := feedback * feedbackMultiplier;

IF setpointFreezeEnable THEN
    setpointTarget := lastSetpoint;
ELSE
    setpointTarget := setpoint * setpointMultiplier;
    IF setpointTarget < setpointMin THEN
        setpointTarget := setpointMin;
    ELSIF setpointTarget > setpointMax THEN
        setpointTarget := setpointMax;
    END_IF;
END_IF;

setpointFrozen := setpointFreezeEnable;
startRamp := FALSE;
deviationMagnitude := setpointTarget - lastSetpointTarget;
IF deviationMagnitude < REAL#0.0 THEN
    deviationMagnitude := -deviationMagnitude;
END_IF;
IF (deviationMagnitude > setpointEpsilon) OR resetEdge THEN
    startRamp := TRUE;
END_IF;
lastSetpointTarget := setpointTarget;

IF (setpointIncreaseTime > T#0S) AND (setpointDecreaseTime > T#0S) THEN
    CASE setpointRampType OF
        RampType#SShaped:
            IF setpointTarget >= lastSetpoint THEN
                remainingTime := setpointIncreaseTime;
            ELSE
                remainingTime := setpointDecreaseTime;
            END_IF;

            sShapedFunc(
                execute := startRamp OR sShapedFunc.busy,
                clock := clock,
                startValue := lastSetpoint,
                endValue := setpointTarget,
                duration := remainingTime,
                tickTime := tickTime
            );

            IF sShapedFunc.error THEN
                setpointInternal := setpointTarget;
            ELSE
                setpointInternal := sShapedFunc.output;
            END_IF;

        RampType#Exponential:
            IF setpointTarget >= lastSetpoint THEN
                remainingTime := setpointIncreaseTime;
            ELSE
                remainingTime := setpointDecreaseTime;
            END_IF;

            delayTicks := UDINT#0;
            WHILE remainingTime > T#0S DO
                delayTicks := delayTicks + UDINT#1;
                IF remainingTime > tickTime THEN
                    remainingTime := remainingTime - tickTime;
                ELSE
                    remainingTime := T#0S;
                END_IF;
            END_WHILE;

            IF delayTicks = UDINT#0 THEN
                deltaTime := REAL#0.001;
            ELSE
                deltaTime := TO_REAL(delayTicks) / REAL#4.605;
                IF deltaTime < REAL#0.001 THEN
                    deltaTime := REAL#0.001;
                END_IF;
            END_IF;

            expRamp(
                execute := TRUE,
                clock := clock,
                reset := startRamp,
                input := setpointTarget,
                T := deltaTime,
                tickTime := tickTime
            );

            IF expRamp.error THEN
                setpointInternal := setpointTarget;
            ELSE
                setpointInternal := expRamp.output;
            END_IF;

        ELSE
            spRange := setpointMax - setpointMin;
            IF spRange < REAL#1.0 THEN
                spRange := REAL#1.0;
            END_IF;

            remainingTime := setpointIncreaseTime;
            increaseTicks := UDINT#0;
            WHILE remainingTime > T#0S DO
                increaseTicks := increaseTicks + UDINT#1;
                IF remainingTime > tickTime THEN
                    remainingTime := remainingTime - tickTime;
                ELSE
                    remainingTime := T#0S;
                END_IF;
            END_WHILE;
            IF increaseTicks = UDINT#0 THEN
                increaseTicks := UDINT#1;
            END_IF;

            remainingTime := setpointDecreaseTime;
            decreaseTicks := UDINT#0;
            WHILE remainingTime > T#0S DO
                decreaseTicks := decreaseTicks + UDINT#1;
                IF remainingTime > tickTime THEN
                    remainingTime := remainingTime - tickTime;
                ELSE
                    remainingTime := T#0S;
                END_IF;
            END_WHILE;
            IF decreaseTicks = UDINT#0 THEN
                decreaseTicks := UDINT#1;
            END_IF;

            setpointInternal := lastSetpoint;
            IF clock THEN
                IF setpointTarget > lastSetpoint THEN
                    rampStep := spRange / TO_REAL(increaseTicks);
                    setpointInternal := lastSetpoint + rampStep;
                    IF setpointInternal > setpointTarget THEN
                        setpointInternal := setpointTarget;
                    END_IF;
                ELSIF setpointTarget < lastSetpoint THEN
                    rampStep := spRange / TO_REAL(decreaseTicks);
                    setpointInternal := lastSetpoint - rampStep;
                    IF setpointInternal < setpointTarget THEN
                        setpointInternal := setpointTarget;
                    END_IF;
                END_IF;
            END_IF;
    END_CASE;
ELSE
    setpointInternal := setpointTarget;
END_IF;

lastSetpoint := setpointInternal;
setpointActual := setpointInternal;

IF deviationInversion THEN
    deviationActual := feedbackActual - setpointActual;
ELSE
    deviationActual := setpointActual - feedbackActual;
END_IF;

deviationMagnitude := deviationActual;
IF deviationMagnitude < REAL#0.0 THEN
    deviationMagnitude := -deviationMagnitude;
END_IF;

remainingTime := deadbandDelay;
delayTicks := UDINT#0;
WHILE remainingTime > T#0S DO
    delayTicks := delayTicks + UDINT#1;
    IF remainingTime > tickTime THEN
        remainingTime := remainingTime - tickTime;
    ELSE
        remainingTime := T#0S;
    END_IF;
END_WHILE;

IF (deadbandRange > REAL#0.0) AND (deviationMagnitude <= deadbandRange) THEN
    IF clock THEN
        deadbandCounter := deadbandCounter + UDINT#1;
    END_IF;
ELSE
    deadbandCounter := UDINT#0;
END_IF;

IF (deadbandRange > REAL#0.0) AND (delayTicks > UDINT#0) AND (deadbandCounter >= delayTicks) THEN
    deadband := TRUE;
ELSE
    deadband := FALSE;
END_IF;

sleepReq := (sleepLevel > REAL#0.0)
    AND (lastPidOutput <= sleepLevel)
    AND (NOT sleepMode)
    AND (NOT sleepBoost)
    AND (NOT trackingMode);

remainingTime := sleepDelay;
delayTicks := UDINT#0;
WHILE remainingTime > T#0S DO
    delayTicks := delayTicks + UDINT#1;
    IF remainingTime > tickTime THEN
        remainingTime := remainingTime - tickTime;
    ELSE
        remainingTime := T#0S;
    END_IF;
END_WHILE;

IF sleepReq THEN
    IF clock THEN
        sleepCounter := sleepCounter + UDINT#1;
    END_IF;
ELSE
    sleepCounter := UDINT#0;
END_IF;

wakeupReq := FALSE;
IF wakeupDeviation > REAL#0.0 THEN
    wakeupReq := (deviationMagnitude >= wakeupDeviation) AND sleepMode;
END_IF;

remainingTime := wakeupDelay;
delayTicks := UDINT#0;
WHILE remainingTime > T#0S DO
    delayTicks := delayTicks + UDINT#1;
    IF remainingTime > tickTime THEN
        remainingTime := remainingTime - tickTime;
    ELSE
        remainingTime := T#0S;
    END_IF;
END_WHILE;

IF wakeupReq THEN
    IF clock THEN
        wakeupCounter := wakeupCounter + UDINT#1;
    END_IF;
ELSE
    wakeupCounter := UDINT#0;
END_IF;

IF (sleepCounter >= delayTicks) AND (sleepReq) AND (delayTicks > UDINT#0) THEN
    sleepCounter := UDINT#0;
    IF (sleepBoostLevel > REAL#0.0) AND (sleepBoostTime > T#0S) THEN
        sleepBoost := TRUE;
    ELSE
        sleepMode := TRUE;
    END_IF;
END_IF;

remainingTime := sleepBoostTime;
delayTicks := UDINT#0;
WHILE remainingTime > T#0S DO
    delayTicks := delayTicks + UDINT#1;
    IF remainingTime > tickTime THEN
        remainingTime := remainingTime - tickTime;
    ELSE
        remainingTime := T#0S;
    END_IF;
END_WHILE;

IF sleepBoost THEN
    IF clock THEN
        sleepBoostCounter := sleepBoostCounter + UDINT#1;
    END_IF;
    IF (delayTicks > UDINT#0) AND (sleepBoostCounter >= delayTicks) THEN
        sleepBoost := FALSE;
        sleepMode := TRUE;
        sleepBoostCounter := UDINT#0;
    END_IF;
ELSE
    sleepBoostCounter := UDINT#0;
END_IF;

IF (delayTicks > UDINT#0) AND (wakeupCounter >= delayTicks) AND wakeupReq THEN
    sleepMode := FALSE;
    sleepBoost := FALSE;
    wakeupCounter := UDINT#0;
    sleepCounter := UDINT#0;
END_IF;

manualMode := FALSE;
yManual := lastOutput;
tracking := FALSE;

IF trackingMode THEN
    tracking := TRUE;
    manualMode := TRUE;
    yManual := trackingRef;
ELSIF sleepBoost THEN
    manualMode := TRUE;
    yManual := sleepBoostLevel;
ELSIF sleepMode THEN
    manualMode := TRUE;
    yManual := REAL#0.0;
ELSIF deadband THEN
    manualMode := TRUE;
    yManual := lastOutput;
ELSIF outputFreezeEnable THEN
    manualMode := TRUE;
    yManual := lastOutput;
END_IF;

remainingTime := tickTime;
delayTicks := UDINT#0;
WHILE remainingTime > T#0S DO
    delayTicks := delayTicks + UDINT#1;
    IF remainingTime > T#1ms THEN
        remainingTime := remainingTime - T#1ms;
    ELSE
        remainingTime := T#0S;
    END_IF;
END_WHILE;
IF delayTicks = UDINT#0 THEN
    deltaTime := REAL#0.01;
ELSE
    deltaTime := TO_REAL(delayTicks) / REAL#1000.0;
END_IF;

rawOutput := previousOutput;
proportionalTerm := REAL#0.0;
derivativeTerm := REAL#0.0;

IF manualMode THEN
    rawOutput := yManual;
ELSE
    IF clock OR resetEdge THEN
        proportionalTerm := gain * deviationActual;

        IF integrationTime > REAL#0.0 THEN
            integralTerm := integralTerm + (gain * deviationActual * deltaTime / integrationTime);
            IF integralTerm > REAL#1000000.0 THEN
                integralTerm := REAL#1000000.0;
                overflow := TRUE;
            ELSIF integralTerm < REAL#-1000000.0 THEN
                integralTerm := REAL#-1000000.0;
                overflow := TRUE;
            END_IF;
        ELSE
            integralTerm := REAL#0.0;
        END_IF;

        IF derivationTime > REAL#0.0 THEN
            deltaDeviation := deviationActual - previousDeviation;
            derivativeTerm := gain * derivationTime * deltaDeviation / deltaTime;
        END_IF;

        rawOutput := offset + proportionalTerm + integralTerm + derivativeTerm;
        previousDeviation := deviationActual;
        previousOutput := rawOutput;
    END_IF;
END_IF;

outputLimitsActive := FALSE;
IF rawOutput < outputMin THEN
    rawOutput := outputMin;
    outputLimitsActive := TRUE;
ELSIF rawOutput > outputMax THEN
    rawOutput := outputMax;
    outputLimitsActive := TRUE;
END_IF;

outputActual := rawOutput;
lastOutput := outputActual;
lastPidOutput := outputActual;
outputFrozen := outputFreezeEnable OR deadband;

zeroOutput := FALSE;
IF outputActual < REAL#0.0 THEN
    IF -outputActual < setpointEpsilon THEN
        zeroOutput := TRUE;
    END_IF;
ELSE
    IF outputActual < setpointEpsilon THEN
        zeroOutput := TRUE;
    END_IF;
END_IF;

atSetpoint := deviationMagnitude < atSetpointHysteresis;
END_FUNCTION_BLOCK

(* ---- R_TRIG.st ---- *)
FUNCTION_BLOCK R_TRIG
VAR_INPUT
    CLK : BOOL;
END_VAR
VAR_OUTPUT
    Q : BOOL;
END_VAR
VAR
    previousClock : BOOL;
END_VAR

Q := CLK AND NOT previousClock;
previousClock := CLK;
END_FUNCTION_BLOCK
